(* IEC 61131-3 sources: FishAndCat/plc (part 2) *)

(* ---- 05_PRG_Main.st ---- *)
(* ============================================================
   05_PRG_Main.st — 主程序(状态机)
   导入方法:POU 类型"程序(Program)",挂到循环任务(建议周期 10ms)
   演示流程(决赛口径):初始化 → 交互输入/载入演示批次 → 批量分配
   → 局部搜索(AWRA-LS)→ 统计 → 可视化呈现;全程非阻塞。
   ============================================================ *)
PROGRAM PRG_Main
VAR
    eState      : E_MainState := E_MainState.STATE_IDLE;
    fbInit      : FB_InitWarehouse;
    fbAssign    : FB_AssignAllGoods;
    fbImprove   : FB_LocalSwapImprove;
    fbStats     : FB_Stats;
    fbPath      : FB_BuildVisuPath;
    fbGoodsInput : FB_GoodsInput;       // 交互货物输入封装(0707 T2.2,替代内联逻辑+fbSelOne)
    fbVisu      : FB_VisuRefresh;       // L6:颜色镜像+堆垛机像素坐标,每周期常驻
    fbAnim      : FB_AnimatePath;       // L6:堆垛机沿路径回放动画(CmdAnimate 触发)
    fbQuery     : FB_QueryGood;         // 块3 P3:单件查询(细则8,常驻)
    fbRecPage   : FB_RecordPage;        // 块3 P2:记录页 10 行窗口(细则8,常驻)
    fbSceneDet  : FB_SceneDetect;       // A2:场景检测器(画像→推荐,常驻自动重算)
    fbAuth      : FB_UserAuth;          // A4:两级权限登录(常驻)
    fbGuard     : FB_ParamGuard;        // A4:调参守卫(常驻,双闸之二)
    xKickInit, xKickAssign, xKickImprove, xKickStats : BOOL;
    xUseRank    : BOOL;
    iStrat      : INT;
    c2, t2      : INT;                  // 清除推荐高亮用循环变量
    xDemoOld, xRunOld, xResetOld : BOOL;
    xSnapOld    : BOOL;                 // 块3:快照按钮沿检测
    xMaintOld   : BOOL;                 // A3:检修按钮沿检测
    iMaintRet   : INT;                  // A3:FC_MaintToggle 返回码
    xViewOld    : BOOL;                 // C2/C6:视图循环按钮沿检测
END_VAR

// ---------- 全局按钮:复位(任意状态可触发) ----------
IF GVL_Visu.CmdReset AND NOT xResetOld THEN
    GVL_WH.iGoodsCount := 0;
    GVL_WH.stStats.PlacedCnt := 0;  GVL_WH.stStats.FailedCnt := 0;
    GVL_Visu.VisuStatusText := 'RESET_INIT';
    GVL_Visu.VisuAlarm := FALSE;                    // 复位清报警灯
    GVL_Visu.VisuPathCount := 0;                    // 复位清路径叠加
    GVL_Visu.VisuCurrentX := 0;                     // 堆垛机归位 I/O 口(左下角)
    GVL_Visu.VisuCurrentY := 0;
    // 0711 修:复位同时清统计/路径显示残留(旧版遗留 186.0/370 等旧批数字误导评委)
    GVL_Visu.VisuTotalTime := 0.0;
    GVL_Visu.VisuAvgTime := 0.0;
    GVL_Visu.VisuSpaceUtilization := 0.0;
    GVL_Visu.VisuWearIndex := 0.0;
    GVL_Visu.VisuViolationCount := 0;
    GVL_Visu.VisuPathLen := 0.0;
    GVL_Visu.VisuExecTime := 0.0;
    GVL_Visu.VisuTargetX := 0;
    GVL_Visu.VisuTargetY := 0;
    eState := E_MainState.STATE_INIT;
END_IF
xResetOld := GVL_Visu.CmdReset;

CASE eState OF
    // ---------- 待机:上电自动进入初始化 ----------
    E_MainState.STATE_IDLE:
        eState := E_MainState.STATE_INIT;

    // ---------- 初始化仓库 ----------
    E_MainState.STATE_INIT:
        xKickInit := TRUE;
        fbInit(xExecute := xKickInit, iRule := GVL_Param.iPreRule);
        IF fbInit.xDone THEN
            xKickInit := FALSE;
            GVL_Visu.VisuStatusText := CONCAT('READY_PRECOUNT=', INT_TO_STRING(fbInit.iPreCount));
            eState := E_MainState.STATE_WAIT_INPUT;
        END_IF

    // ---------- 等待输入(决赛交互:逐件添加 / 载入演示批 / 启动批量) ----------
    E_MainState.STATE_WAIT_INPUT:
        // 按钮1:添加单件货物(五属性)——逻辑封装进 FB_GoodsInput(0707 T2.2),PRG 只编排可视化
        fbGoodsInput(xAdd := GVL_Visu.CmdAddGood,
                     iId := GVL_Visu.InGoodId, sName := GVL_Visu.InGoodName,
                     rWeight := GVL_Visu.InGoodWeight, rFreq := GVL_Visu.InGoodFreq,
                     rVolume := GVL_Visu.InGoodVolume);
        IF fbGoodsInput.xOk THEN
            IF fbGoodsInput.xFound THEN
                GVL_Visu.VisuSlotState[fbGoodsInput.iSugX, fbGoodsInput.iSugY] := 3;  // 黄:推荐
                fbPath(xExecute := TRUE,  iToX := fbGoodsInput.iSugX, iToY := fbGoodsInput.iSugY);
                fbPath(xExecute := FALSE, iToX := fbGoodsInput.iSugX, iToY := fbGoodsInput.iSugY);
                GVL_Visu.VisuStatusText := CONCAT('SUGGEST_X=',
                    CONCAT(INT_TO_STRING(fbGoodsInput.iSugX),
                    CONCAT('_Y=', INT_TO_STRING(fbGoodsInput.iSugY))));
                GVL_Visu.VisuAlarm := FALSE;                   // 推荐成功清报警灯
            ELSE
                GVL_Visu.VisuStatusText := 'ALARM_NO_FEASIBLE_SLOT';   // 边界#9 超重货无位
                GVL_Visu.VisuAlarm := TRUE;                    // 红灯(演示第6步)
            END_IF
        ELSIF fbGoodsInput.iErrId = 1 THEN
            GVL_Visu.VisuStatusText := 'ERR_GOODS_FULL_400';   // 边界:满仓
            GVL_Visu.VisuAlarm := TRUE;
        ELSIF fbGoodsInput.iErrId = 2 THEN
            GVL_Visu.VisuStatusText := 'ERR_NEG_INPUT';        // 边界:负输入
            GVL_Visu.VisuAlarm := TRUE;
        END_IF

        // 按钮2:载入演示批次(GVL_Data,由 Python seed=2026 导出,保证与仿真同源)
        IF GVL_Visu.CmdLoadDemo AND NOT xDemoOld THEN
            FC_LoadDemoGoods();
            GVL_Visu.VisuStatusText := CONCAT('DEMO_LOADED_N=',
                                              INT_TO_STRING(GVL_WH.iGoodsCount));
            GVL_Visu.VisuAlarm := FALSE;                // 新批次开始,清报警灯与旧路径
            GVL_Visu.VisuPathCount := 0;
        END_IF
        xDemoOld := GVL_Visu.CmdLoadDemo;

        // 按钮3:运行批量分配
        IF GVL_Visu.CmdRunAssign AND NOT xRunOld THEN
            IF GVL_WH.iGoodsCount = 0 THEN
                GVL_Visu.VisuStatusText := 'ERR_NO_GOODS';
                GVL_Visu.VisuAlarm := TRUE;
            ELSE
                // 进入批量前清交互阶段残留:推荐黄格回写空闲(推荐只会盖在空闲格上,
                // fbSelOne 只选可行空位,故直接回写0安全)+ 路径叠加清除 + 报警灯灭
                FOR c2 := 0 TO GVL_Param.COLS - 1 DO
                    FOR t2 := 0 TO GVL_Param.TIERS - 1 DO
                        IF GVL_Visu.VisuSlotState[c2, t2] = 3 THEN
                            GVL_Visu.VisuSlotState[c2, t2] := 0;
                        END_IF
                    END_FOR
                END_FOR
                GVL_Visu.VisuPathCount := 0;
                GVL_Visu.VisuAlarm := FALSE;
                // 策略选择:0=seq 1=near 2=score(在线) 3=AWRA-LS(批量=Rank+score+LS)
                xUseRank := (GVL_Visu.SelStrategy = 3);
                IF GVL_Visu.SelStrategy = 3 THEN iStrat := 2; ELSE iStrat := GVL_Visu.SelStrategy; END_IF
                xKickAssign := TRUE;
                eState := E_MainState.STATE_ASSIGN;
            END_IF
        END_IF
        xRunOld := GVL_Visu.CmdRunAssign;

    // ---------- 批量分配(分片运行中) ----------
    E_MainState.STATE_ASSIGN:
        fbAssign(xStart := xKickAssign, xUseRank := xUseRank, iStrategy := iStrat);
        xKickAssign := FALSE;
        GVL_Visu.VisuStatusText := CONCAT('ASSIGN_RUN_PLACED=', INT_TO_STRING(fbAssign.iAssigned));
        IF fbAssign.xDone THEN
            IF GVL_Visu.SelStrategy = 3 THEN
                xKickImprove := TRUE;
                eState := E_MainState.STATE_IMPROVE;
            ELSE
                xKickStats := TRUE;
                eState := E_MainState.STATE_STATS;
            END_IF
        END_IF

    // ---------- 局部搜索(仅 AWRA-LS,分片运行中) ----------
    E_MainState.STATE_IMPROVE:
        fbImprove(xStart := xKickImprove);
        xKickImprove := FALSE;
        GVL_Visu.VisuStatusText := CONCAT('IMPROVE_R=',
            CONCAT(INT_TO_STRING(fbImprove.iRounds),
            CONCAT('_SWAPS=', INT_TO_STRING(fbImprove.iSwaps))));
        IF fbImprove.xDone THEN
            GVL_WH.stStats.SwapCnt  := fbImprove.iSwaps;
            GVL_WH.stStats.LsRounds := fbImprove.iRounds;
            xKickStats := TRUE;
            eState := E_MainState.STATE_STATS;
        END_IF

    // ---------- 统计 ----------
    E_MainState.STATE_STATS:
        fbStats(xExecute := xKickStats);
        xKickStats := FALSE;
        IF fbStats.xDone THEN
            GVL_Visu.VisuWearIndex := GVL_WH.stStats.PathTotal2Way;   // 损耗代理=路径总长(C5)
            eState := E_MainState.STATE_DONE;
        END_IF

    // ---------- 完成:结果驻留可视化;失败件数非0则警示文本+红灯 ----------
    E_MainState.STATE_DONE:
        IF GVL_WH.stStats.FailedCnt > 0 THEN
            GVL_Visu.VisuStatusText := CONCAT('DONE_FAILED_N=',
                                              INT_TO_STRING(GVL_WH.stStats.FailedCnt));
            GVL_Visu.VisuAlarm := TRUE;    // 与其他异常态一致:有货无位=红灯(0705补)
        ELSE
            GVL_Visu.VisuStatusText := 'DONE_OK';
        END_IF
        // 停留本状态;CmdReset 重来(顶部全局处理)

    E_MainState.STATE_FAULT:
        ;   // 预留:严重故障驻留(当前边界均以文本报警+拒绝操作处理)
END_CASE

// ---------- L6 常驻段(每周期,与状态机无关) ----------
// 块3 P2/P3:记录页窗口+单件查询(常驻:DONE 后评委翻表/查询仍可用)
fbRecPage(xPageUp := GVL_Visu.CmdPageUp, xPageDown := GVL_Visu.CmdPageDown);
fbQuery(xQuery := GVL_Visu.CmdQuery, iId := GVL_Visu.InQueryId);
// A2 场景检测器:货物表变化自动重算画像+推荐;Auto 开=推荐直写策略档(人工覆盖=关 Auto)
fbSceneDet();
IF fbSceneDet.xValid AND GVL_Visu.xAutoStrategy THEN
    GVL_Visu.SelStrategy := fbSceneDet.iRecBatch;
END_IF
// A4 登录/登出+调参守卫;PIN 消费即清(登录动作当周期已用,不留回显/重放)
fbAuth(xLogin := GVL_Visu.CmdLogin, iPin := GVL_Visu.InPinCode,
       xLogout := GVL_Visu.CmdLogout);
GVL_Visu.iUserLevel := fbAuth.iLevel;
GVL_Visu.VisuUserText := fbAuth.sUserText;
IF GVL_Visu.CmdLogin OR GVL_Visu.CmdLogout THEN
    GVL_Visu.InPinCode := 0;
END_IF
fbGuard(iLevel := fbAuth.iLevel);
// A3 检修挂起/恢复(需管理员;putaway block 语义:禁新入库,存量冻结可查询)
IF GVL_Visu.CmdMaintToggle AND NOT xMaintOld THEN
    iMaintRet := FC_MaintToggle(x := GVL_Visu.InMaintX, y := GVL_Visu.InMaintY,
                                iLevel := fbAuth.iLevel);
    CASE iMaintRet OF
        0: GVL_Visu.VisuStatusText := CONCAT('MAINT_SET_X=',
               CONCAT(INT_TO_STRING(GVL_Visu.InMaintX),
               CONCAT('_Y=', INT_TO_STRING(GVL_Visu.InMaintY))));
        1: GVL_Visu.VisuStatusText := CONCAT('MAINT_CLR_X=',
               CONCAT(INT_TO_STRING(GVL_Visu.InMaintX),
               CONCAT('_Y=', INT_TO_STRING(GVL_Visu.InMaintY))));
        2: GVL_Visu.VisuStatusText := 'ERR_MAINT_NEED_ADMIN';
        3: GVL_Visu.VisuStatusText := 'ERR_MAINT_RANGE';
    END_CASE
END_IF
xMaintOld := GVL_Visu.CmdMaintToggle;
// C2/C6 视图循环:状态→频次热力→损耗热力→状态(操作员可用,分析视图)
IF GVL_Visu.CmdViewCycle AND NOT xViewOld THEN
    GVL_Visu.iViewMode := (GVL_Visu.iViewMode + 1) MOD 3;
    CASE GVL_Visu.iViewMode OF
        0: GVL_Visu.VisuStatusText := 'VIEW_STATE';
        1: GVL_Visu.VisuStatusText := 'VIEW_HEAT_FREQ';
        2: GVL_Visu.VisuStatusText := 'VIEW_HEAT_WEAR';
    END_CASE
END_IF
xViewOld := GVL_Visu.CmdViewCycle;
// 块3 方向9:快照保存(上升沿把当前布局冻结为对比基准,CmdCompareMode 切换显示)
IF GVL_Visu.CmdSaveSnap AND NOT xSnapOld THEN
    GVL_Visu.aSnapState := GVL_Visu.VisuSlotState;      // 同型数组整体赋值
    GVL_Visu.xSnapValid := TRUE;
    GVL_Visu.VisuStatusText := 'SNAP_SAVED';
END_IF
xSnapOld := GVL_Visu.CmdSaveSnap;
// 块3:名称下拉同步(ComboBox 写入下标,消费即复位=一次性写入不锁手输)
IF GVL_Visu.iNameSel >= 0 AND GVL_Visu.iNameSel <= 9 THEN
    GVL_Visu.InGoodName := GVL_Visu.astrNames[GVL_Visu.iNameSel];
    GVL_Visu.iNameSel := -1;
END_IF
// 动画回放:CmdAnimate 上升沿触发,堆垛机图元沿当前 VisuPath 走到目标格
// (rCycleTime 与本任务周期一致:10ms 任务填 0.01;改任务周期须同步这里)
fbAnim(xStart := GVL_Visu.CmdAnimate, rCycleTime := 0.01, rSpeedScale := 5.0);
// ---------- 0711 疫苗:脉冲命令消费即复位(段尾,所有消费者已跑完) ----------
// 防两类实测事故:①MouseUp 事件丢失致命令卡 TRUE(Load demo 风暴 N=260)
// ②输入积压在 download 后突发重放。复位后命令只存活一个扫描周期,天然免疫。
// 注意:CmdCompareMode/xAutoStrategy 是翻转开关、SelStrategy 是 INT 档位,均不得复位。
GVL_Visu.CmdAddGood   := FALSE;
GVL_Visu.CmdLoadDemo  := FALSE;
GVL_Visu.CmdRunAssign := FALSE;
GVL_Visu.CmdReset     := FALSE;
GVL_Visu.CmdAnimate   := FALSE;
GVL_Visu.CmdSaveSnap  := FALSE;
GVL_Visu.CmdQuery     := FALSE;
GVL_Visu.CmdPageUp    := FALSE;
GVL_Visu.CmdPageDown  := FALSE;
GVL_Visu.CmdLogin     := FALSE;     // A4(0711)
GVL_Visu.CmdLogout    := FALSE;
GVL_Visu.CmdMaintToggle := FALSE;   // A3(0711)
GVL_Visu.CmdViewCycle := FALSE;     // C2/C6(0711;iViewMode 是档位、InTierSel 是数值,均不复位)
// 颜色镜像+堆垛机像素坐标刷新(画面所有动态元件的数据源,必须在 fbAnim 之后)
fbVisu();
END_PROGRAM

(* ---- 06_PRG_Test.st ---- *)
(* ============================================================
   06_PRG_Test.st — 边界与一致性测试程序
   导入方法:POU 类型"程序",可挂到同一任务或手动调用;
   置 xRunTests:=TRUE 单次运行,看 iPassed/iFailed/aResult。
   覆盖:资料包 §7.3 边界判断清单 + Python↔ST 评分一致性向量 + B1 官方口径(T24)
   (向量由 sim/export_st_vectors.py 生成于 07_GVL_Data_generated.st,
    与仿真同源 —— 这是"PLC 实现与验证报告数字互相背书"的证据链)
   注意:测试会改写仓库状态,跑完请按 CmdReset 重新初始化再演示。
   ============================================================ *)
PROGRAM PRG_Test
VAR
    xRunTests : BOOL;                       // 置 TRUE 触发(自动复位)
    iPassed   : INT;
    iFailed   : INT;
    xAllPass  : BOOL;
    N_CASES   : INT := 59;                  // 用例总数(0711 A2-A4 T46-56;C1/C2/C6 T57-59)
    aResult   : ARRAY[1..59] OF BOOL;       // 各用例结果(TRUE=通过)
    sLastFail : STRING[64];                 // 最后失败的用例名(排错入口)
    fbInit    : FB_InitWarehouse;
    fbSel     : FB_SelectSlot;
    fbAssign  : FB_AssignAllGoods;          // T25 端到端:AWRA 分配状态机
    fbImprove : FB_LocalSwapImprove;        // T25 端到端:局部搜索状态机
    fbStats   : FB_Stats;                   // T25 端到端:终局统计
    fbGoodsInputT : FB_GoodsInput;          // T41:货物输入封装测试
    fbQueryT  : FB_QueryGood;               // T42:单件查询测试(块3)
    fbRecPageT : FB_RecordPage;             // T43:记录页窗口测试(块3)
    fbDetT    : FB_SceneDetect;             // T49-T53:场景检测器测试(A2,0711)
    fbAuthT   : FB_UserAuth;                // T54:两级权限测试(A4,0711)
    fbGuardT  : FB_ParamGuard;              // T55:调参守卫测试(A4,0711)
    fbVisuT   : FB_VisuRefresh;             // T59:层高亮/层计数测试(C1,0711)
    iRet      : INT;                        // T56:FC_MaintToggle 返回码
    dwBefore  : DWORD;                      // T59:高亮前色值(相对锚)
    i, x, y, n : INT;
    rV        : REAL;
    iVecFail  : INT;
    iAwraPosDiff : INT;                     // T25 逐位分歧计数(信息性;0=终局布局与 sim 逐位一致)
END_VAR

IF xRunTests THEN
    xRunTests := FALSE;
    iPassed := 0;  iFailed := 0;  sLastFail := '';
    FOR i := 1 TO 59 DO aResult[i] := TRUE; END_FOR

    // ---- T01-T04 承重系数:正常/顶层/负钳位/越上钳位 ----
    aResult[1] := ABS(FC_CapCoef(y := 0)  - 1.0)  < 0.0001;
    aResult[2] := ABS(FC_CapCoef(y := 19) - 0.62) < 0.0001;
    aResult[3] := ABS(FC_CapCoef(y := -5) - 1.0)  < 0.0001;
    aResult[4] := ABS(FC_CapCoef(y := 25) - 0.62) < 0.0001;

    // ---- T05-T07 预占用历史三解读格数(49/231/134;官方口径 sum 见 T24) ----
    n := 0;
    FOR x := 0 TO 19 DO FOR y := 0 TO 19 DO
        IF FC_IsPresetOccupied(x := x, y := y, iRule := 0) THEN n := n + 1; END_IF
    END_FOR END_FOR
    aResult[5] := (n = 49);
    n := 0;
    FOR x := 0 TO 19 DO FOR y := 0 TO 19 DO
        IF FC_IsPresetOccupied(x := x, y := y, iRule := 1) THEN n := n + 1; END_IF
    END_FOR END_FOR
    aResult[6] := (n = 231);
    n := 0;
    FOR x := 0 TO 19 DO FOR y := 0 TO 19 DO
        IF FC_IsPresetOccupied(x := x, y := y, iRule := 2) THEN n := n + 1; END_IF
    END_FOR END_FOR
    aResult[7] := (n = 134);

    // ---- T08-T10 行程时间双模型 + 路径长度(vx=2.0, vy=0.5 时的已知值) ----
    rV := FC_CalcTravelTime(x0 := 0, y0 := 0, x1 := 19, y1 := 19, xSimXY := TRUE);
    aResult[8] := ABS(rV - 38.0) < 0.001;                       // 切比雪夫 max(9.5, 38)
    rV := FC_CalcTravelTime(x0 := 0, y0 := 0, x1 := 19, y1 := 19, xSimXY := FALSE);
    aResult[9] := ABS(rV - 47.5) < 0.001;                       // 顺序 9.5+38
    aResult[10] := ABS(FC_CalcPathLen(x0 := 0, y0 := 0, x1 := 19, y1 := 19) - 38.0) < 0.001;

    // ---- 初始化仓库(rule=0),供可行性/选位用例使用 ----
    fbInit(xExecute := FALSE, iRule := 0);
    fbInit(xExecute := TRUE,  iRule := 0);

    // ---- T11-T16 可行性边界:正常/预占/超重/负重/超容/越界 ----
    aResult[11] :=      FC_CheckFeasible(x := 1,  y := 0,  rGoodW := 80.0, rGoodV := 0.5);
    aResult[12] := NOT  FC_CheckFeasible(x := 0,  y := 0,  rGoodW := 10.0, rGoodV := 0.5);  // (0,0)预占
    aResult[13] := NOT  FC_CheckFeasible(x := 1,  y := 10, rGoodW := 81.0, rGoodV := 0.5);  // cap=80
    aResult[14] := NOT  FC_CheckFeasible(x := 1,  y := 0,  rGoodW := -1.0, rGoodV := 0.5);
    aResult[15] := NOT  FC_CheckFeasible(x := 1,  y := 0,  rGoodW := 10.0, rGoodV := 1.2);
    aResult[16] := NOT  FC_CheckFeasible(x := 20, y := 0,  rGoodW := 10.0, rGoodV := 0.5);

    // ---- T17 超重货全库无可行位(>100kg 连底层都放不下) ----
    fbSel(iStrategy := 2, rGoodW := 150.0, rGoodF := 50.0, rGoodV := 0.5,
          rWMax := 150.0, rFMax := 100.0);
    aResult[17] := NOT fbSel.xFound;

    // ---- T18 满仓无可行位(边界#所有仓位已满) ----
    FOR x := 0 TO 19 DO FOR y := 0 TO 19 DO
        GVL_WH.aSlots[x, y].Occupied := TRUE;
    END_FOR END_FOR
    fbSel(iStrategy := 2, rGoodW := 10.0, rGoodF := 1.0, rGoodV := 0.5,
          rWMax := 10.0, rFMax := 1.0);
    aResult[18] := NOT fbSel.xFound;
    fbInit(xExecute := FALSE, iRule := 0);          // 恢复
    fbInit(xExecute := TRUE,  iRule := 0);

    // ---- T19 评分一致性向量(Python 导出,容差1e-3;见 07_GVL_Data_generated.st) ----
    iVecFail := 0;
    FOR i := 1 TO GVL_Data.N_TESTVEC DO
        rV := FC_CalcScore(rGoodW := GVL_Data.aTestVec[i].W,
                           rGoodF := GVL_Data.aTestVec[i].F,
                           x := GVL_Data.aTestVec[i].X, y := GVL_Data.aTestVec[i].Y,
                           rWMax := GVL_Data.aTestVec[i].WMax,
                           rFMax := GVL_Data.aTestVec[i].FMax);
        IF ABS(rV - GVL_Data.aTestVec[i].ExpScore) >= 0.001 THEN
            iVecFail := iVecFail + 1;
        END_IF
    END_FOR
    aResult[19] := (iVecFail = 0);

    // ---- T20 行程时间一致性向量(同上) ----
    iVecFail := 0;
    FOR i := 1 TO GVL_Data.N_TESTVEC DO
        rV := FC_CalcTravelTime(x0 := 0, y0 := 0,
                                x1 := GVL_Data.aTestVec[i].X, y1 := GVL_Data.aTestVec[i].Y,
                                xSimXY := TRUE);
        IF ABS(rV - GVL_Data.aTestVec[i].ExpTime) >= 0.001 THEN
            iVecFail := iVecFail + 1;
        END_IF
    END_FOR
    aResult[20] := (iVecFail = 0);

    // ---- T21 演示批次载入自检(件数与来源标记) ----
    GVL_WH.iGoodsCount := 0;
    FC_LoadDemoGoods();
    aResult[21] := (GVL_WH.iGoodsCount = GVL_Data.N_DEMO);

    // ---- T22 L1 加减速口径一致性向量(与 Python 梯形模型逐条比对) ----
    GVL_Param.xUseAccel := TRUE;
    iVecFail := 0;
    FOR i := 1 TO GVL_Data.N_TESTVEC DO
        rV := FC_CalcTravelTime(x0 := 0, y0 := 0,
                                x1 := GVL_Data.aTestVec[i].X, y1 := GVL_Data.aTestVec[i].Y,
                                xSimXY := TRUE);
        IF ABS(rV - GVL_Data.aTestVec[i].ExpTimeAccel) >= 0.001 THEN
            iVecFail := iVecFail + 1;
        END_IF
    END_FOR
    GVL_Param.xUseAccel := FALSE;               // 恢复默认口径
    aResult[22] := (iVecFail = 0);

    // ---- T23 双命令周期:已知值 + 不劣于单命令(C10) ----
    // 存(5,2) 取(10,5),匀速切比雪夫:t存=max(2.5,4)=4, t间=max(2.5,6)=6, t取=max(5,10)=10
    rV := FC_CalcDualCycleTime(iStoreX := 5, iStoreY := 2, iRetrX := 10, iRetrY := 5);
    aResult[23] := (ABS(rV - 20.0) < 0.001)
                   AND (rV <= 2.0 * 4.0 + 2.0 * 10.0 + 0.001);

    // ---- T24 B1 官方口径(2026-07-06 答复):x+y 之和被3整除 = 133 格 ----
    // 官方原话"x+y 和能被3整除";含 (0,0) 格,呈对角条纹;与 Python 侧
    // test_preoccupied_counts 的 sum=133 断言同口径(双实现同步铁律)
    n := 0;
    FOR x := 0 TO 19 DO FOR y := 0 TO 19 DO
        IF FC_IsPresetOccupied(x := x, y := y, iRule := 3) THEN n := n + 1; END_IF
    END_FOR END_FOR
    aResult[24] := (n = 133);

    // ---- T25 AWRA-LS 全流程终局一致性(端到端护栏;0707,sim/consistency_probe 离线证明可绿) ----
    // 驱动 Rank+Assign+LS 分片状态机跑到 xDone(WHILE 内推进,测试不计实时性),
    // 比对终局:①聚合统计容差(主判据,对单双精度局部最优鲁棒,同 T19/T20 哲学)
    //          ②终局布局逐位(信息性 iAwraPosDiff;G1/G2 零触发时应为 0,见 gap 表)
    // 向量源:07_GVL_Data_generated.st 的 aAwraExpect / AWRA_EXPT/ENERGY/COG(sum 官方口径,匀速)
    GVL_Param.xUseAccel := FALSE;                    // 与 export 同口径(匀速)
    GVL_WH.iGoodsCount := 0;
    fbInit(xExecute := FALSE, iRule := 3);
    fbInit(xExecute := TRUE,  iRule := 3);           // sum 官方口径(133 预占)
    FC_LoadDemoGoods();                              // 20 件 seed2026,与 sim 同源
    // -- 驱动 AWRA 分配(xUseRank=TRUE 排序模式,score 策略=2) --
    fbAssign(xStart := FALSE, xUseRank := TRUE, iStrategy := 2);
    fbAssign(xStart := TRUE,  xUseRank := TRUE, iStrategy := 2);
    n := 0;
    WHILE fbAssign.xBusy AND (n < 100000) DO
        fbAssign(xStart := TRUE, xUseRank := TRUE, iStrategy := 2);
        n := n + 1;
    END_WHILE
    // -- 驱动局部搜索到收敛 --
    fbImprove(xStart := FALSE);
    fbImprove(xStart := TRUE);
    n := 0;
    WHILE fbImprove.xBusy AND (n < 1000000) DO
        fbImprove(xStart := TRUE);
        n := n + 1;
    END_WHILE
    // -- 终局统计 --
    fbStats(xExecute := FALSE);
    fbStats(xExecute := TRUE);
    // -- 逐位信息性检查(aGoods 索引==Id,见 FC_LoadDemoGoods) --
    iAwraPosDiff := 0;
    FOR i := 1 TO GVL_Data.N_AWRA DO
        IF (GVL_WH.aGoods[GVL_Data.aAwraExpect[i].Id].X <> GVL_Data.aAwraExpect[i].X)
        OR (GVL_WH.aGoods[GVL_Data.aAwraExpect[i].Id].Y <> GVL_Data.aAwraExpect[i].Y) THEN
            iAwraPosDiff := iAwraPosDiff + 1;
        END_IF
    END_FOR
    // -- 主判据:逐位一致(演示批 consistency_probe 证 G1/G2 零触发,故逐位可作主判据)
    //    + 聚合容差 + 计数精确 + 违规0(多重护栏) --
    aResult[25] := (iAwraPosDiff = 0)
       AND (GVL_WH.stStats.PlacedCnt = GVL_Data.AWRA_PLACED)
       AND (GVL_WH.stStats.FailedCnt = GVL_Data.AWRA_FAILED)
       AND (ABS(GVL_WH.stStats.ExpRetrieval - GVL_Data.AWRA_EXPT) < 0.001)
       AND (ABS(GVL_WH.stStats.Energy      - GVL_Data.AWRA_ENERGY) < 0.01)
       AND (ABS(GVL_WH.stStats.CogHeight   - GVL_Data.AWRA_COG) < 0.001)
       AND (GVL_WH.stStats.ViolCnt = 0);

    // ---- T26-T35 边界判断扩充(0707,评分细则5"边界判断充分";纯函数断言,手算期望) ----
    // 重置干净仓库(T25 跑满;and 口径 rule0 供边界测试,MaxWeight[y]=CapCoef(y)*100)
    GVL_WH.iGoodsCount := 0;
    fbInit(xExecute := FALSE, iRule := 0);
    fbInit(xExecute := TRUE,  iRule := 0);
    GVL_Param.xUseAccel := FALSE;
    // T26-T27 坐标越界(FC_CheckFeasible 显式范围检查,先于数组访问,不靠 CheckBounds 钳位)
    aResult[26] := NOT FC_CheckFeasible(x := -1, y := 0,  rGoodW := 10.0, rGoodV := 0.5);  // 负列
    aResult[27] := NOT FC_CheckFeasible(x := 0,  y := 20, rGoodW := 10.0, rGoodV := 0.5);  // 越层(y>19)
    // T28-T29 负属性(显式拒绝)
    aResult[28] := NOT FC_CheckFeasible(x := 5, y := 0, rGoodW := -1.0, rGoodV := 0.5);    // 负重
    aResult[29] := NOT FC_CheckFeasible(x := 5, y := 0, rGoodW := 10.0, rGoodV := -0.1);   // 负容
    // T30-T31 承重边界(y=10 限重80/y=19 限重62;留 0.1 间隙避单精度噪声)
    aResult[30] :=     FC_CheckFeasible(x := 1, y := 10, rGoodW := 79.9, rGoodV := 0.5)
               AND NOT FC_CheckFeasible(x := 1, y := 10, rGoodW := 80.1, rGoodV := 0.5);
    aResult[31] :=     FC_CheckFeasible(x := 1, y := 19, rGoodW := 61.9, rGoodV := 0.5)
               AND NOT FC_CheckFeasible(x := 1, y := 19, rGoodW := 62.1, rGoodV := 0.5);
    // T32 容积边界(CELL_VOL=1.0)
    aResult[32] :=     FC_CheckFeasible(x := 1, y := 0, rGoodW := 10.0, rGoodV := 0.99)
               AND NOT FC_CheckFeasible(x := 1, y := 0, rGoodW := 10.0, rGoodV := 1.01);
    // T33-T34 归一分母为0保护(不除零崩溃,返回有限非负;枪I:REAL除零=INF/NaN 依系统)
    rV := FC_CalcScore(rGoodW := 10.0, rGoodF := 5.0, x := 1, y := 0, rWMax := 0.0, rFMax := 0.0);
    // 归一保护后 rFMax→1、F=5>1 使 fNorm=5、resv=(1-5)*.. 为负,score 可负——本用例只验
    // "除零保护生效=返回有限值不崩"(NaN 令两比较皆 FALSE、INF 令 <1E6 FALSE,故此区间≡有限数)
    aResult[33] := (rV > -1.0E6) AND (rV < 1.0E6);
    rV := FC_CalcPriority(rGoodF := 5.0, rGoodW := 10.0, rGoodV := 0.5,
                          rFMax := 0.0, rWMax := 0.0, rVMax := 0.0);
    aResult[34] := (rV >= 0.0) AND (rV < 100.0);
    // T35 优先级单调性(同重同体积,高频→优先级更高;Rank 阶段正确性)
    aResult[35] := FC_CalcPriority(rGoodF := 100.0, rGoodW := 10.0, rGoodV := 0.5,
                                   rFMax := 100.0, rWMax := 100.0, rVMax := 1.0)
                 > FC_CalcPriority(rGoodF := 1.0, rGoodW := 10.0, rGoodV := 0.5,
                                   rFMax := 100.0, rWMax := 100.0, rVMax := 1.0);

    // ---- T36-T40 选位策略边界(0707;FB_SelectSlot 各策略正确性;仓库=上面 rule0 干净态) ----
    // T36 seq 策略:首个可行位((0,0)预占 → 扫描到 (0,1))
    fbSel(iStrategy := 0, rGoodW := 10.0, rGoodF := 5.0, rGoodV := 0.5, rWMax := 10.0, rFMax := 5.0);
    aResult[36] := fbSel.xFound AND (fbSel.iBestX = 0) AND (fbSel.iBestY = 1);
    // T37 near 策略:行程时间最小可行位((1,0) travel=max(0.5,0)=0.5 全库最小)
    fbSel(iStrategy := 1, rGoodW := 10.0, rGoodF := 5.0, rGoodV := 0.5, rWMax := 10.0, rFMax := 5.0);
    aResult[37] := fbSel.xFound AND (fbSel.iBestX = 1) AND (fbSel.iBestY = 0);
    // T38 score 策略:有解(多目标评分选位)
    fbSel(iStrategy := 2, rGoodW := 10.0, rGoodF := 5.0, rGoodV := 0.5, rWMax := 10.0, rFMax := 5.0);
    aResult[38] := fbSel.xFound;
    // T39 中重货 90kg 只能进低层(限重≥90 → 层 y≤5),仍有解
    fbSel(iStrategy := 1, rGoodW := 90.0, rGoodF := 5.0, rGoodV := 0.5, rWMax := 90.0, rFMax := 5.0);
    aResult[39] := fbSel.xFound AND (fbSel.iBestY <= 5);
    // T40 FB_SelectSlot 无副作用:同输入重复调用结果一致(纯功能,只读仓库)
    fbSel(iStrategy := 2, rGoodW := 25.0, rGoodF := 8.0, rGoodV := 0.5, rWMax := 25.0, rFMax := 8.0);
    x := fbSel.iBestX;  y := fbSel.iBestY;
    fbSel(iStrategy := 2, rGoodW := 25.0, rGoodF := 8.0, rGoodV := 0.5, rWMax := 25.0, rFMax := 8.0);
    aResult[40] := (fbSel.iBestX = x) AND (fbSel.iBestY = y);

    // ---- T41 FB_GoodsInput 封装(评分细则6/7;0707 T2.2 抽取):正常/负输入/超重无位 三分支 ----
    GVL_WH.iGoodsCount := 0;
    fbInit(xExecute := FALSE, iRule := 0);
    fbInit(xExecute := TRUE,  iRule := 0);
    // (a) 正常轻货 → xOk & xFound & 入表(count=1)
    fbGoodsInputT(xAdd := FALSE, iId := 1, sName := 'A', rWeight := 10.0, rFreq := 5.0, rVolume := 0.5);
    fbGoodsInputT(xAdd := TRUE,  iId := 1, sName := 'A', rWeight := 10.0, rFreq := 5.0, rVolume := 0.5);
    aResult[41] := fbGoodsInputT.xOk AND fbGoodsInputT.xFound AND (GVL_WH.iGoodsCount = 1);
    // (b) 负输入 → 拒收 iErrId=2,不入表(count 仍 1;新上升沿=先落再起)
    fbGoodsInputT(xAdd := FALSE, iId := 2, sName := 'B', rWeight := -1.0, rFreq := 5.0, rVolume := 0.5);
    fbGoodsInputT(xAdd := TRUE,  iId := 2, sName := 'B', rWeight := -1.0, rFreq := 5.0, rVolume := 0.5);
    aResult[41] := aResult[41] AND (NOT fbGoodsInputT.xOk) AND (fbGoodsInputT.iErrId = 2)
                   AND (GVL_WH.iGoodsCount = 1);
    // (c) 超重货 150kg → 入表但无可行位 iErrId=3、xFound=FALSE(新上升沿)
    fbGoodsInputT(xAdd := FALSE, iId := 3, sName := 'C', rWeight := 150.0, rFreq := 5.0, rVolume := 0.5);
    fbGoodsInputT(xAdd := TRUE,  iId := 3, sName := 'C', rWeight := 150.0, rFreq := 5.0, rVolume := 0.5);
    aResult[41] := aResult[41] AND fbGoodsInputT.xOk AND (NOT fbGoodsInputT.xFound)
                   AND (fbGoodsInputT.iErrId = 3);

    // ---- T42-T45 块3 画面服务(0708;前置=T41 留下的表:aGoods[1]=Id1轻货/aGoods[2]=Id3超重,count=2) ----
    GVL_Param.xUseAccel := FALSE;           // 测试自给自足:显式匀速口径(防前序用例遗留开关)
    GVL_Param.xSimultaneousXY := TRUE;      // 同上:显式切比雪夫主口径(T42 拟真锚 7.5s 依赖)

    // T42 FB_QueryGood:未分配/已分配+高亮+拟真字段/未找到清旧高亮/非正Id 四分支
    // (a) 未分配货:找得到,属性对,位置=-1
    fbQueryT(xQuery := FALSE, iId := 1);
    fbQueryT(xQuery := TRUE,  iId := 1);
    aResult[42] := GVL_Visu.QryFound AND (ABS(GVL_Visu.QryWeight - 10.0) < 0.001)
                   AND (GVL_Visu.QryX = -1);
    // (b) 手工落位 (2,3) 再查:位置/路径/高亮/拟真对照全齐
    //     手算锚:laden(0,0→2,3)=MAX(2/2, 3/(0.5×0.8))=MAX(1.0,7.5)=7.5s;10kg→轻档 6.0s
    GVL_WH.aGoods[1].Assigned := TRUE;
    GVL_WH.aGoods[1].X := 2;   GVL_WH.aGoods[1].Y := 3;
    GVL_WH.aGoods[1].PathLength := 5.0;  GVL_WH.aGoods[1].ExecTime := 6.0;
    fbQueryT(xQuery := FALSE, iId := 1);
    fbQueryT(xQuery := TRUE,  iId := 1);
    aResult[42] := aResult[42] AND GVL_Visu.QryFound
                   AND (GVL_Visu.QryX = 2) AND (GVL_Visu.QryY = 3)
                   AND (ABS(GVL_Visu.QryPathLen - 5.0) < 0.001)
                   AND (GVL_Visu.VisuSlotState[2, 3] = 6)
                   AND (ABS(GVL_Visu.QryTravelLaden - 7.5) < 0.001)
                   AND (ABS(GVL_Visu.QryHandleT - 6.0) < 0.001);
    // (c) 查不存在 Id:Found=FALSE 且旧青色高亮恢复为已占用 2
    fbQueryT(xQuery := FALSE, iId := 999);
    fbQueryT(xQuery := TRUE,  iId := 999);
    aResult[42] := aResult[42] AND (NOT GVL_Visu.QryFound)
                   AND (GVL_Visu.VisuSlotState[2, 3] = 2);
    // (d) 非正 Id:直接未找到(边界)
    fbQueryT(xQuery := FALSE, iId := -1);
    fbQueryT(xQuery := TRUE,  iId := -1);
    aResult[42] := aResult[42] AND (NOT GVL_Visu.QryFound);

    // T43 FB_RecordPage:窗口映射/空行约定/小表钳位/大表翻页钳位
    // (a) 2 件小表:顶行=1,行0=Id1(已落位 X=2),行1=Id3(未分配 X=-1),行2=空(Id=0)
    fbRecPageT(xPageUp := FALSE, xPageDown := FALSE);
    aResult[43] := (GVL_Visu.iRecTop = 1) AND (GVL_Visu.aRowId[0] = 1)
                   AND (GVL_Visu.aRowX[0] = 2) AND (GVL_Visu.aRowId[1] = 3)
                   AND (GVL_Visu.aRowX[1] = -1) AND (GVL_Visu.aRowId[2] = 0)
                   AND (GVL_Visu.iRecTotal = 2);
    // (b) 小表下翻:钳位拉回 1(2 件表无第二页)
    fbRecPageT(xPageUp := FALSE, xPageDown := TRUE);
    aResult[43] := aResult[43] AND (GVL_Visu.iRecTop = 1);
    // (c) 造 25 件大表验证翻页链:1→11→16(25-9 钳位)→6(上翻);毕恢复 count=2
    GVL_WH.iGoodsCount := 25;
    fbRecPageT(xPageUp := FALSE, xPageDown := FALSE);   // 沿复位
    fbRecPageT(xPageUp := FALSE, xPageDown := TRUE);
    aResult[43] := aResult[43] AND (GVL_Visu.iRecTop = 11);
    fbRecPageT(xPageUp := FALSE, xPageDown := FALSE);
    fbRecPageT(xPageUp := FALSE, xPageDown := TRUE);
    aResult[43] := aResult[43] AND (GVL_Visu.iRecTop = 16);
    fbRecPageT(xPageUp := FALSE, xPageDown := FALSE);
    fbRecPageT(xPageUp := TRUE,  xPageDown := FALSE);
    aResult[43] := aResult[43] AND (GVL_Visu.iRecTop = 6);
    GVL_WH.iGoodsCount := 2;

    // T44 FC_HandleTime 三档边界(0.1 间隙避单精度,块2 惯例):29.9轻/30.1中/60.0中含/60.1重
    aResult[44] := (ABS(FC_HandleTime(rW := 29.9) - 6.0)  < 0.001)
                   AND (ABS(FC_HandleTime(rW := 30.1) - 8.5)  < 0.001)
                   AND (ABS(FC_HandleTime(rW := 60.0) - 8.5)  < 0.001)
                   AND (ABS(FC_HandleTime(rW := 60.1) - 12.5) < 0.001);

    // T45 FC_TravelLaden:垂直折减/水平不折减/顺序分支/非法系数保护
    // 手算锚(匀速):laden(0,0→10,10)切比雪夫=MAX(10/2, 10/0.4)=25.0(空载同点=20.0)
    aResult[45] := (ABS(FC_TravelLaden(x0:=0, y0:=0, x1:=10, y1:=10, xSimXY:=TRUE) - 25.0) < 0.001)
                   AND (ABS(FC_CalcTravelTime(x0:=0, y0:=0, x1:=10, y1:=10, xSimXY:=TRUE) - 20.0) < 0.001);
    // 水平纯移动:折减只作用垂直 → 与空载同值 5.0
    aResult[45] := aResult[45]
                   AND (ABS(FC_TravelLaden(x0:=0, y0:=0, x1:=10, y1:=0, xSimXY:=TRUE) - 5.0) < 0.001);
    // 顺序模型分支:5+25=30.0
    aResult[45] := aResult[45]
                   AND (ABS(FC_TravelLaden(x0:=0, y0:=0, x1:=10, y1:=10, xSimXY:=FALSE) - 30.0) < 0.001);
    // 非法折减系数保护:0.0 → 不折减(=空载 20.0);毕恢复默认 0.80
    GVL_Param.rLadenFactorVY := 0.0;
    aResult[45] := aResult[45]
                   AND (ABS(FC_TravelLaden(x0:=0, y0:=0, x1:=10, y1:=10, xSimXY:=TRUE) - 20.0) < 0.001);
    GVL_Param.rLadenFactorVY := 0.80;

    // ============ 0711 A2-A4:T46-T56(检修挂起/场景检测器/两级权限) ============

    // ---- T46-T48 检修挂起(A3,putaway block 语义;干净仓:sum 口径 133 预占) ----
    fbInit(xExecute := FALSE, iRule := 3);
    fbInit(xExecute := TRUE,  iRule := 3);
    // T46 挂起→选位不可行;恢复→立即回池(挂起/恢复双向)
    GVL_WH.aMaintBlock[1, 0] := TRUE;
    aResult[46] := NOT FC_CheckFeasible(x := 1, y := 0, rGoodW := 10.0, rGoodV := 0.5);
    GVL_WH.aMaintBlock[1, 0] := FALSE;
    aResult[46] := aResult[46]
                   AND FC_CheckFeasible(x := 1, y := 0, rGoodW := 10.0, rGoodV := 0.5);
    // T47 集成:near 轻货首选 (1,0)(t=0.5s);挂起后绕行次优 (2,0)(t=1.0s);恢复后回 (1,0)
    GVL_WH.aMaintBlock[1, 0] := TRUE;
    fbSel(iStrategy := 1, rGoodW := 10.0, rGoodF := 50.0, rGoodV := 0.5,
          rWMax := 100.0, rFMax := 100.0);
    aResult[47] := fbSel.xFound AND (fbSel.iBestX = 2) AND (fbSel.iBestY = 0);
    GVL_WH.aMaintBlock[1, 0] := FALSE;
    fbSel(iStrategy := 1, rGoodW := 10.0, rGoodF := 50.0, rGoodV := 0.5,
          rWMax := 100.0, rFMax := 100.0);
    aResult[47] := aResult[47] AND fbSel.xFound AND (fbSel.iBestX = 1) AND (fbSel.iBestY = 0);
    // T48 交换目标位检修=禁入(FC_FitsPhysical;检修位存量可换走、新货不得换进)
    GVL_WH.aMaintBlock[2, 0] := TRUE;
    aResult[48] := NOT FC_FitsPhysical(x := 2, y := 0, rGoodW := 10.0, rGoodV := 0.5);
    GVL_WH.aMaintBlock[2, 0] := FALSE;
    aResult[48] := aResult[48]
                   AND FC_FitsPhysical(x := 2, y := 0, rGoodW := 10.0, rGoodV := 0.5);

    // ---- T49-T53 场景检测器(A2;画像手算锚+推荐分支全覆盖) ----
    // 5 件手工批:freq 10/20/30/40/100(和=200),w 10/20/30/70/80 → n=5;
    // density=5/267=0.018727;top=MAX(1,5/5)=1 件 → skew=100/200=0.5;
    // w_mean=210/5=42.0;w_heavy(>60kg)=2/5=0.4
    FOR i := 1 TO 5 DO
        GVL_WH.aGoods[i].Id := i;  GVL_WH.aGoods[i].Volume := 0.5;
        GVL_WH.aGoods[i].Assigned := FALSE;
    END_FOR
    GVL_WH.aGoods[1].Freq := 10.0;   GVL_WH.aGoods[1].Weight := 10.0;
    GVL_WH.aGoods[2].Freq := 20.0;   GVL_WH.aGoods[2].Weight := 20.0;
    GVL_WH.aGoods[3].Freq := 30.0;   GVL_WH.aGoods[3].Weight := 30.0;
    GVL_WH.aGoods[4].Freq := 40.0;   GVL_WH.aGoods[4].Weight := 70.0;
    GVL_WH.aGoods[5].Freq := 100.0;  GVL_WH.aGoods[5].Weight := 80.0;
    GVL_WH.iGoodsCount := 5;
    FOR i := 1 TO 10 DO fbDetT(xForce := FALSE); IF fbDetT.xValid THEN EXIT; END_IF END_FOR
    // T49 画像位级(容差 1e-3,块2 一致性惯例)
    aResult[49] := fbDetT.xValid
                   AND (GVL_Visu.VisuProfN = 5)
                   AND (ABS(GVL_Visu.VisuProfDensity - 0.018727) < 0.001)
                   AND (ABS(GVL_Visu.VisuProfSkew - 0.5) < 0.001)
                   AND (ABS(GVL_Visu.VisuProfWMean - 42.0) < 0.001)
                   AND (ABS(GVL_Visu.VisuProfWHeavy - 0.4) < 0.001);
    // T50 批量推荐:skew 0.5>=0.35 → AWRA(holistic 全要素档)
    aResult[50] := (fbDetT.iRecBatch = 3);
    // T51 在线推荐:n=5<=20 → near(F18-2 极小批降级)
    aResult[51] := (fbDetT.iRecOnline = 1);
    // T52 均匀批(freq 全 50→skew=0.2<0.35 且 n<=20):批量/在线均 near;xForce 重算路径
    FOR i := 1 TO 5 DO GVL_WH.aGoods[i].Freq := 50.0; END_FOR
    fbDetT(xForce := FALSE);
    FOR i := 1 TO 10 DO fbDetT(xForce := TRUE); IF fbDetT.xValid THEN EXIT; END_IF END_FOR
    aResult[52] := fbDetT.xValid AND (fbDetT.iRecBatch = 1) AND (fbDetT.iRecOnline = 1)
                   AND (ABS(GVL_Visu.VisuProfSkew - 0.2) < 0.001);
    // T53 大批高偏(n=21>20,skew=(100+10*3)/300=0.4333>=0.35):批量 AWRA/在线 score
    FOR i := 1 TO 20 DO
        GVL_WH.aGoods[i].Id := i;      GVL_WH.aGoods[i].Freq := 10.0;
        GVL_WH.aGoods[i].Weight := 50.0;  GVL_WH.aGoods[i].Volume := 0.5;
    END_FOR
    GVL_WH.aGoods[21].Id := 21;  GVL_WH.aGoods[21].Freq := 100.0;
    GVL_WH.aGoods[21].Weight := 50.0;  GVL_WH.aGoods[21].Volume := 0.5;
    GVL_WH.iGoodsCount := 21;
    FOR i := 1 TO 10 DO fbDetT(xForce := FALSE); IF fbDetT.xValid THEN EXIT; END_IF END_FOR
    aResult[53] := fbDetT.xValid AND (fbDetT.iRecBatch = 3) AND (fbDetT.iRecOnline = 2)
                   AND (ABS(GVL_Visu.VisuProfSkew - 0.43333) < 0.001);
    GVL_WH.iGoodsCount := 2;                        // 对齐 T43 尾惯例,防状态外溢

    // ---- T54-T55 两级权限(A4:登录三段 + 守卫回滚) ----
    // T54 错码拒登(计数+1)→ 对码升管理员 → 登出回操作员
    fbAuthT(xLogin := FALSE, iPin := 0, xLogout := FALSE);
    fbAuthT(xLogin := TRUE,  iPin := 1111, xLogout := FALSE);
    aResult[54] := (fbAuthT.iLevel = 0) AND (fbAuthT.iFailCnt = 1);
    fbAuthT(xLogin := FALSE, iPin := 0, xLogout := FALSE);
    fbAuthT(xLogin := TRUE,  iPin := GVL_Param.ADMIN_PIN, xLogout := FALSE);
    aResult[54] := aResult[54] AND (fbAuthT.iLevel = 1);
    fbAuthT(xLogin := FALSE, iPin := 0, xLogout := TRUE);
    aResult[54] := aResult[54] AND (fbAuthT.iLevel = 0);
    // T55 守卫:管理员改参被保持;操作员级越权改动一周期内回滚
    fbGuardT(iLevel := 1);                          // 首 call:快照=现值(0.15)
    GVL_Param.rDelta := 0.99;                       // 管理员改参
    fbGuardT(iLevel := 1);                          // 快照刷新=0.99
    fbGuardT(iLevel := 0);                          // 降级:合法值保持
    aResult[55] := (ABS(GVL_Param.rDelta - 0.99) < 0.001);
    GVL_Param.rDelta := 0.5;                        // 操作员越权改
    fbGuardT(iLevel := 0);                          // 守卫回滚到 0.99
    aResult[55] := aResult[55] AND (ABS(GVL_Param.rDelta - 0.99) < 0.001);
    GVL_Param.rDelta := 0.15;                       // 恢复默认并刷快照(防外溢)
    fbGuardT(iLevel := 1);

    // ---- T56 检修权限门(FC_MaintToggle 四分支:需管理员/挂起/恢复/越界) ----
    n := GVL_Visu.VisuMaintCount;                   // 相对基准(在线演示可能已有检修格)
    iRet := FC_MaintToggle(x := 5, y := 5, iLevel := 0);
    aResult[56] := (iRet = 2) AND NOT GVL_WH.aMaintBlock[5, 5];
    iRet := FC_MaintToggle(x := 5, y := 5, iLevel := 1);
    aResult[56] := aResult[56] AND (iRet = 0) AND GVL_WH.aMaintBlock[5, 5]
                   AND (GVL_Visu.VisuMaintCount = n + 1);
    iRet := FC_MaintToggle(x := 5, y := 5, iLevel := 1);
    aResult[56] := aResult[56] AND (iRet = 1) AND NOT GVL_WH.aMaintBlock[5, 5]
                   AND (GVL_Visu.VisuMaintCount = n);
    iRet := FC_MaintToggle(x := -1, y := 0, iLevel := 1);
    aResult[56] := aResult[56] AND (iRet = 3);

    // ============ 0711 C1/C2/C6:T57-T59(热力色阶/仓位履历/层高亮) ============

    // ---- T57 FC_HeatColor 三段端点 + 防除 + FC_BlendLight 黑白极值(手算锚) ----
    aResult[57] := (FC_HeatColor(rVal := 0.0,   rMax := 100.0) = DWORD#16#FF1565C0)
               AND (FC_HeatColor(rVal := 50.0,  rMax := 100.0) = DWORD#16#FFFFD600)
               AND (FC_HeatColor(rVal := 100.0, rMax := 100.0) = DWORD#16#FFE53935)
               AND (FC_HeatColor(rVal := 5.0,   rMax := 0.0)   = DWORD#16#FF1565C0)
               AND (FC_BlendLight(dw := DWORD#16#FF000000) = DWORD#16#FF737373)
               AND (FC_BlendLight(dw := DWORD#16#FFFFFFFF) = DWORD#16#FFFFFFFF);

    // ---- T58 aSlotOps 履历 + aSlotFreq 布局态(小批端到端:2 件 score 落位) ----
    fbInit(xExecute := FALSE, iRule := 3);
    fbInit(xExecute := TRUE,  iRule := 3);              // aSlotFreq 随批清;aSlotOps 履历保留
    aResult[58] := (ABS(GVL_WH.aSlotFreq[10, 10]) < 0.0001);   // init 后布局态干净
    GVL_WH.aGoods[1].Id := 1;  GVL_WH.aGoods[1].Weight := 10.0;
    GVL_WH.aGoods[1].Freq := 5.0;  GVL_WH.aGoods[1].Volume := 0.5;
    GVL_WH.aGoods[1].Assigned := FALSE;
    GVL_WH.aGoods[2].Id := 2;  GVL_WH.aGoods[2].Weight := 20.0;
    GVL_WH.aGoods[2].Freq := 3.0;  GVL_WH.aGoods[2].Volume := 0.5;
    GVL_WH.aGoods[2].Assigned := FALSE;
    GVL_WH.iGoodsCount := 2;
    fbAssign(xStart := FALSE, xUseRank := FALSE, iStrategy := 2);
    fbAssign(xStart := TRUE,  xUseRank := FALSE, iStrategy := 2);
    n := 0;
    WHILE fbAssign.xBusy AND (n < 100000) DO
        fbAssign(xStart := TRUE, xUseRank := FALSE, iStrategy := 2);
        n := n + 1;
    END_WHILE
    aResult[58] := aResult[58] AND GVL_WH.aGoods[1].Assigned
               AND (ABS(GVL_WH.aSlotFreq[GVL_WH.aGoods[1].X, GVL_WH.aGoods[1].Y] - 5.0) < 0.0001)
               AND (GVL_WH.aSlotOps[GVL_WH.aGoods[1].X, GVL_WH.aGoods[1].Y] >= 1)
               AND (GVL_WH.aSlotOps[GVL_WH.aGoods[2].X, GVL_WH.aGoods[2].Y] >= 1);

    // ---- T59 层高亮集成:计数正确 + 高亮色=FC_BlendLight(原色)(相对锚,免猜状态色) ----
    GVL_Visu.InTierSel := -1;
    fbVisuT();                                          // 无高亮基准帧
    x := GVL_WH.aGoods[1].X;  y := GVL_WH.aGoods[1].Y;
    dwBefore := GVL_Visu.VisuSlotColor[x, GVL_Param.TIERS - 1 - y];
    aResult[59] := (GVL_Visu.VisuTierOcc = 0);
    GVL_Visu.InTierSel := y;
    fbVisuT();                                          // 高亮该层
    aResult[59] := aResult[59] AND (GVL_Visu.VisuTierOcc >= 1)
               AND (GVL_Visu.VisuSlotColor[x, GVL_Param.TIERS - 1 - y]
                    = FC_BlendLight(dw := dwBefore));
    GVL_Visu.InTierSel := -1;                           // 恢复,防外溢
    GVL_WH.iGoodsCount := 2;

    // ---- 汇总 ----
    FOR i := 1 TO N_CASES DO
        IF aResult[i] THEN iPassed := iPassed + 1;
        ELSE
            iFailed := iFailed + 1;
            sLastFail := CONCAT('T', INT_TO_STRING(i));
        END_IF
    END_FOR
    xAllPass := (iFailed = 0);
END_IF
END_PROGRAM
